TYPE SAI_InputRealChannel :
STRUCT
	{attribute addProperty Name "Value"}
	Value AT %I* : REAL;
END_STRUCT
END_TYPE

(* stored: Version 1.1.0.1, ProductVersion 3.1.4024.9
   DUT SAI_InputRealChannel: Id {f6343b2d-fe3f-0782-3522-cbc8994840c4} *)
